{attribute 'qualified_only'}
// GENERATED FILE — DO NOT EDIT. §8.8/§8.9 catalog size.
VAR_GLOBAL CONSTANT
    COUNT : INT := 63;
END_VAR

(* stored: Version 1.1.0.1, ProductVersion 3.1.4024.12
   GVL PL_ReasonCatalog: Id {51b77bda-8d2b-4dad-9187-16d040699e35} *)
